(*udt (user defined type) for all EtherCAT Based Trumpf Laser Interfacing on EL6692, up to 64 Bytes
	Author(S): Justin Vandongen of Sodecia GTAC;

------------------------------------------------------------------------
	REVISION NOTES:

	Version 20171002
		- Initial Concept, j.vandongen

------------------------------------------------------------------------
*)



TYPE udt_EtherCat_Trumpf_InputWords_20171002 :
STRUCT
	Laser_Out: ARRAY [0..9] OF WORD;
END_STRUCT
END_TYPE

(* stored: Version 1.1.0.1, ProductVersion 3.1.4024.5
   DUT udt_EtherCat_Trumpf_InputWords_20171002: Id {0ee7ccf1-fd45-49a9-bdb9-463c50176e8c} *)
